// TIA Portal V20 export
TYPE "Udt_M200D_OUT"
   STRUCT
      "Motor CW" : Bool;
      "Motor CCW" : Bool;
      "Control for brake" : Bool;
      "Trip reset" : Bool;
      "Emergency start" : Bool;
      "Self-test" : Bool;
      Unassigned1 : Bool;
      Unassigned2 : Bool;
      "Output 1" : Bool;
      "Output 2" : Bool;
      Unassigned3 : Bool;
      Unassigned4 : Bool;
      Unassigned5 : Bool;
      Unassigned6 : Bool;
      Unassigned7 : Bool;
      "Disable quick stop" : Bool;
   END_STRUCT;
END_TYPE
